{attribute 'qualified_only'}
VAR_GLOBAL CONSTANT
	MAX_STATIONS	: USINT := 10;
END_VAR

(* stored: Version 1.1.0.1
   GVL CONST: Id {a6f7558e-7310-4080-a423-e00692c98531}, ParameterList True *)
